TYPE ST_Item :
STRUCT
	ID : STRING := '';		// Bar Code 	
	UniqueID : DINT := 0;		// Generic ID for tracking
	Destination : DINT := 0;
	Length : DINT := 0;
	Status : E_StatusCode := E_StatusCode.No_Status;
	ExtStatus : E_StatusCode := E_StatusCode.No_Status;
	CapturedInMetrics : BOOL;
	DeviceID:	STRING(5);	// Device ID associated with this record
	MessageType:	E_MessageIds;	// Message Type associated with this record
END_STRUCT
END_TYPE

(* stored: Version 1.1.0.1, ProductVersion 3.1.4024.4
   DUT ST_Item: Id {5d791c6b-b28c-4c54-9380-14b2cb3fa533} *)
